FUNCTION_BLOCK ABSTRACT AliasDatatypeBase EXTENDS DatatypeBase 
VAR
	baseType : I_Datatype;
END_VAR

METHOD FB_init : BOOL
VAR_INPUT
	bInitRetains : BOOL; // if TRUE, the retain variables are initialized (warm start / cold start)
	bInCopyCode : BOOL;  // if TRUE, the instance afterwards gets moved into the copy code (online change)
END_VAR
InitializeBaseType(baseType);
END_METHOD

PROPERTY PUBLIC ABSTRACT Identifier : T_MAXSTRING
GET
END_GET
END_PROPERTY

PROPERTY PUBLIC IecType : T_MAXSTRING
GET
IecType := 'ALIAS';
END_GET
END_PROPERTY

METHOD PROTECTED ABSTRACT InitializeBaseType
VAR_INPUT
	BaseType : REFERENCE TO I_Datatype;
END_VAR
END_METHOD

METHOD PUBLIC SerializeTypeWith
VAR_INPUT
	Serializer : I_Serializer;
END_VAR
Serializer.StartObject();
Serializer.AddKeyString('name',Identifier);
Serializer.AddKeyString('type',IecType);
Serializer.AddKey('baseType');
baseType.SerializeTypeWith(Serializer);
Serializer.EndObject();
END_METHOD

METHOD PUBLIC SerializeWith
VAR_INPUT
	Serializer : I_Serializer;
END_VAR
Serializer.StartObject();
baseType.SerializeWith(Serializer);
Serializer.EndObject();
END_METHOD

METHOD TryDeserializeFrom : BOOL
VAR_INPUT
	Deserializer : I_Deserializer;
END_VAR
TryDeserializeFrom := baseType.TryDeserializeFrom(Deserializer);
END_METHOD

END_FUNCTION_BLOCK

(* stored: Version 1.1.0.1, ProductVersion 3.1.4024.12
   POU AliasDatatypeBase: Id {51efc251-d562-035f-0714-2cb40d22bd49}, SpecialFunc None
   Folder Constructor: Id {b8636ece-804d-4aef-b7e9-10aa4c674f58}
   Folder Protected: Id {bf24f291-342d-43fe-95fb-0541a5caab0a}
   Method FB_init: Id {b5ef8675-b621-498f-afec-0be9b1011dfb}
   Property Identifier: Id {3a1b6a1c-2ed1-4f30-b499-6a6e905bbab5}
   Get Get: Id {cac64592-d854-4fdc-8853-dc04b5c5a68c}
   Property IecType: Id {4522de90-f1b5-0fc0-0e0b-23cb79104913}
   Get Get: Id {87e770ed-14bd-0fd2-0898-258431f34b50}
   Method InitializeBaseType: Id {c08c071f-acb6-4574-a8aa-fdec38b44307}
   Method SerializeTypeWith: Id {854505f5-1017-462d-a584-80f93779a559}
   Method SerializeWith: Id {0e1207a2-8592-4c4b-9710-52ccdb73d294}
   Method TryDeserializeFrom: Id {d02555e8-a46e-47c3-9f23-7110e9393468} *)
